TYPE T_List_Node : ST_LIST_NODE; END_TYPE

(* stored: Version 1.1.0.1
   DUT T_List_Node: Id {820f3930-feac-0a03-1f4a-f34f8359ce38} *)
